// TIA Portal V17 export
DATA_BLOCK "Conveyor_DB"   // DB3
// stored: InstanceOfName Conveyor, InstanceOfType FB
"Conveyor"
BEGIN
END_DATA_BLOCK
